FUNCTION_BLOCK ConveyorSC
VAR_OUTPUT
	//operation : ConveyorMode;
	
	error AT %I* : BOOL;
	position AT %I* : REAL;
	velocity AT %I* : REAL;
END_VAR
VAR
	enable AT %Q* : BOOL := TRUE;
	direction AT %Q* : BOOL; //FALSE = forward, TRUE = backward
	pulse AT %Q* : BOOL;
	reset AT %Q* : BOOL;
	
	sensorEntry AT %I* : BOOL := TRUE;
	sensorExit AT %I* : BOOL;
END_VAR
VAR
	nextConveyor : POINTER TO ConveyorSC;
	prevConveyor : POINTER TO ConveyorSC;
	
	modeActual : (IDLE, FORWARD, BACKWARD, STOP);
	modeRequest : (IDLE, FORWARD, BACKWARD, STOP);
	
	pulser : TP; //pulses are assumed to be low-high-low
END_VAR
VAR_STAT
	chainRequest : (IDLE, FORWARD, BACKWARD, STOP);
	chainingActive : BOOL; //1st runthrough
	chainingSet : BOOL; //2nd runthrough
END_VAR
VAR_STAT CONSTANT
	pulseWidth : TIME := T#50MS;
END_VAR

override();

sequence();

METHOD backward : BOOL
VAR_INPUT
END_VAR
END_METHOD

METHOD PROTECTED calculateChains : BOOL
VAR_INPUT
END_VAR
IF IsOccupied THEN //chain calculation not started, and this conveyor can start a chain
	chainRequest := MAX(chainRequest, modeRequest);
ELSE
	chainRequest := IDLE;
END_IF

modeActual := chainRequest;
END_METHOD

METHOD forward : BOOL
VAR_INPUT
END_VAR
END_METHOD

{attribute 'monitoring' := 'call'}
PROPERTY IsOccupied : BOOL
GET
IsOccupied := sensorExit OR sensorEntry;
END_GET
END_PROPERTY

METHOD join : BOOL
VAR_INPUT
	conveyor : POINTER TO ConveyorSC;
END_VAR
nextConveyor := conveyor;
conveyor^.prevConveyor := THIS;
END_METHOD

METHOD PROTECTED override : BOOL
VAR_INPUT
END_VAR
(*
IF
	(extended AND lifterMode = UP) OR
	(retracted AND lifterMode = DOWN)
THEN
	lifterMode := HOLD;
END_IF
*)
END_METHOD

METHOD reset : BOOL
VAR_INPUT
END_VAR
position := 0;
velocity := velocity; //no change
END_METHOD

METHOD resetChain : BOOL
VAR_INPUT
END_VAR
chainRequest := 0;
END_METHOD

METHOD PROTECTED sequence : BOOL
VAR_INPUT
END_VAR
calculateChains();

direction := (modeActual = BACKWARD); //set direction bit

pulser(IN:= , PT:= pulseWidth, Q=> pulse, ET=> );
pulser.IN := 
	enable AND 
	NOT error AND 
	NOT reset AND 
	(modeActual = FORWARD OR modeActual = BACKWARD)
	AND pulser.Q; //ends pulse itself
END_METHOD

METHOD target : BOOL
VAR_INPUT
	targetPosition : REAL;
END_VAR
END_METHOD

END_FUNCTION_BLOCK

(* stored: Version 1.1.0.1, ProductVersion 3.1.4024.11
   POU ConveyorSC: Id {860d94bc-eccd-41d5-99ab-6eff761fea1e}, SpecialFunc None
   Folder Private: Id {1ece495e-bdcc-4502-a200-3f9c921872ce}
   Folder Properties: Id {a232f22b-9224-4f1d-a749-173222abc541}
   Folder Unused: Id {54c4b87f-27c9-43c3-88a4-4690df509a73}
   Method backward: Id {68c61c83-5cc5-4351-8ae1-c9fd5871add9}
   Method calculateChains: Id {8af2a1c6-e9d2-4563-8b97-019e5bbfd0c9}
   Method forward: Id {bb5a5b6b-58ec-4b84-83e1-5306f144be0a}
   Property IsOccupied: Id {b654cb6e-3eb6-4615-b963-e01922160291}
   Get Get: Id {fae71c9d-fa89-4510-b5a4-5f3a8d5bd641}
   Method join: Id {4a1ffc9b-791a-4361-acf4-9a8749188615}
   Method override: Id {cb73f434-8629-4f8a-a7be-6a43c7bd04bc}
   Method reset: Id {fc1c874d-d1ec-4894-bc7f-b003bf23e601}
   Method resetChain: Id {f7b73ab0-351e-4e8c-99d7-b0f3f8acb003}
   Method sequence: Id {3852c593-4a74-4095-9f31-2f16a2071246}
   Method target: Id {140af314-e43a-4751-b875-e59fd73378df} *)
